INTERFACE ITF_BaseLogger_Item

METHOD GetInformationToDisplayEvent : ST_BaseLogger_ItemDataToDisplay
VAR_INPUT
	uiIDEvent				: UINT;
END_VAR
END_METHOD

END_INTERFACE

(* stored: Version 1.1.0.1
   Itf ITF_BaseLogger_Item: Id {9acb94a3-79f9-0d22-1a7a-50b9e1991d9a}
   Method GetInformationToDisplayEvent: Id {93fc010a-fb9f-082f-1e1f-a9126d7f1608} *)
